(* IEC 61131-3 sources: tbswQsort/, 3 files *)

(* ---- Quicksort.typ ---- *)
(********************************************************************
 * COPYRIGHT --
 ********************************************************************
 * Library: Quicksort
 * File: Quicksort.typ
 * Author: wielando
 * Created: May 14, 2009
 ********************************************************************
 * Data types of library Quicksort
 ********************************************************************)

TYPE

END_TYPE

(* ---- Quicksort.fun ---- *)
(********************************************************************
 * COPYRIGHT --
 ********************************************************************
 * Library: Quicksort
 * File: Quicksort.fun
 * Author: wielando
 * Created: May 14, 2009
 ********************************************************************
 * Functions and function blocks of library Quicksort
 ********************************************************************)

FUNCTION qsort_str : UINT (*Sortiert Strings mit dem Quicksort-Algorithmus*)
	VAR_INPUT
		pStrings : UDINT; (*Addres of stringarray*)
		len : UDINT; (*Length of one string*)
		count : UDINT; (*Count of strings to sort*)
	END_VAR
END_FUNCTION

FUNCTION qsort_int : UINT (*Sortiert Integer in aufsteigender Reihefolge*)
	VAR_INPUT
		pIntArray : UDINT; (*Add your parameter comment*)
		count : UDINT;
	END_VAR
END_FUNCTION

(* ---- Quicksort.var ---- *)
(********************************************************************
 * COPYRIGHT --
 ********************************************************************
 * Library: Quicksort
 * File: Quicksort.var
 * Author: wielando
 * Created: May 14, 2009
 ********************************************************************
 * Constants of library Quicksort
 ********************************************************************)

VAR CONSTANT

END_VAR
